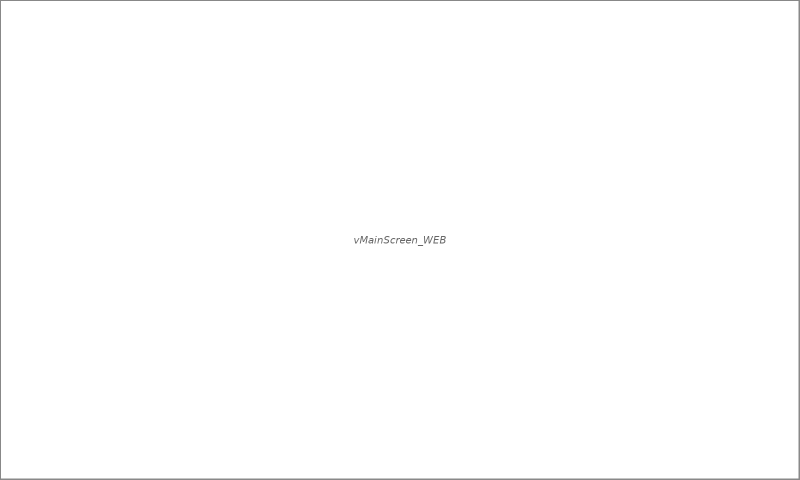
VISUALIZATION vMain_WEB  // 800x480
    Frame (0,0 800x480)
        shows vMainScreen_WEB(arChamber := MAIN.fb.arFbChamber, arParams := GVL_TesterParams.arstParams, arControl := GVL_TesterParams.arstControl, arTestParams := GVL_TesterParams.arTestParams)
        shows vService(fbChamber := arChamber[iActualChamber], stParams := arParams[iActualChamber])
        shows vFileSave(fbChamber := arChamber[iActualChamber], stParams := arParams[iActualChamber])
        shows vPlotScreen(stControl := arControl[iActualChamber], fbChamber := arChamber[iActualChamber])
        shows vStatusScreen_v2(arChamber := arChamber[iActualChamber], arParams := arParams[iActualChamber], arControl := arControl[iActualChamber])
        p2772295162: GVL_TesterParams.arTestParams
        p3795463443: GVL_TesterParams.arstControl
        p1849057978: GVL_TesterParams.arstParams
        p1287185654: MAIN.fb.arFbChamber
END_VISUALIZATION

(* stored: Version 1.1.0.1, ProductVersion 3.1.4024.12
   Visu vMain_WEB: Id {10fef3eb-abad-48b5-aec0-820d3d04917b} *)
